Yaskawa INFORM job: X2_50&56B(90_180).JBI

/JOB
//NAME X2_50&56B(90_180)
//POS
///NPOS 380,380,380,17,0,0
///TOOL 0
///POSTYPE PULSE
///PULSE
C00000=45487,-81749,-76140,5313,88955,-2714
C00001=100725,-66680,-65098,5325,101088,31571
C00002=134065,-13803,-33339,15050,117611,54074
C00003=178572,20950,5765,5105,121785,76071
C00004=178477,15787,3727,4983,120398,75966
C00005=178438,13766,2992,4934,119816,75923
C00006=178435,14063,4928,4877,118781,75875
C00007=178438,13766,2992,4934,119816,75923
C00008=180168,17754,7052,5608,119256,76587
C00009=180168,18141,9405,5533,118013,76523
C00010=179359,16071,7488,5217,118182,76212
C00011=180168,18141,9405,5533,118013,76523
C00012=172189,10953,2801,14884,115134,86218
C00013=173139,8005,189,15209,115045,86581
C00014=172189,10953,2801,14884,115134,86218
C00015=169290,3234,-9196,14399,118965,85580
C00016=130973,-13523,-33423,14333,118859,53260
C00017=110700,-69385,-63067,6190,97747,34870
C00018=68653,-71679,-73408,24733,95794,85842
C00019=66615,-75998,-75470,24709,95531,75346
C00020=80537,-29900,-12555,12207,96591,80441
C00021=81172,-32243,-10721,12278,94215,80425
C00022=81559,-32147,-8308,12330,92754,80411
C00023=81559,-31652,-7175,12323,92320,80369
C00024=79890,-31226,-7999,11978,93276,79895
C00025=78854,-29246,-5136,11740,92696,79487
C00026=78019,-31526,-6644,11553,92575,79192
C00027=78854,-29246,-5136,11740,92696,79487
C00028=78535,-28461,-4244,11667,92599,79369
C00029=79905,-29828,-5160,11964,92267,79802
C00030=78535,-28461,-4244,11667,92599,79369
C00031=80655,-29539,-12313,12233,96610,80484
C00032=172905,9069,10368,17661,103953,63205
C00033=172925,6453,11622,17490,101927,62911
C00034=172953,5852,13232,17402,100678,62738
C00035=172980,6410,14735,17366,100062,62659
C00036=172934,5478,12205,17429,101103,62793
C00037=174868,12262,20269,17776,99277,63224
C00038=175653,10008,18253,17959,99184,63493
C00039=174868,12262,20269,17776,99277,63224
C00040=175466,10534,19114,17901,98978,63395
C00041=174549,8650,17530,17692,99183,63095
C00042=175466,10534,19114,17901,98978,63395
C00043=175364,13912,17144,18083,101810,63784
C00044=143557,-6058,-8183,20909,99706,63742
C00045=116076,-21395,-35361,8294,99864,-41660
C00046=116170,-16904,-19810,8141,92666,-42104
C00047=120850,-15711,-13213,8164,88779,-40753
C00048=120850,-15320,-11697,8164,88052,-40800
C00049=120850,-15603,-12792,8164,88575,-40767
C00050=118682,-15547,-12749,8147,88797,-41494
C00051=118682,-15195,-11396,8147,88151,-41535
C00052=119909,-15242,-11433,8154,88024,-41123
C00053=118283,-15171,-11379,8139,88193,-41669
C00054=118283,-17130,-20118,8163,92522,-41388
C00055=123081,10517,-9626,8350,99710,-39267
C00056=125078,45057,28923,8216,93591,-38991
C00057=129546,52045,50715,11678,83315,-38263
C00058=130769,54168,55563,11090,81346,-37992
C00059=131361,55704,59445,11868,79480,-38000
C00060=131361,56824,62095,11904,78446,-38101
C00061=127122,55959,62427,19640,78177,-40212
C00062=127429,56070,62553,19642,78085,-40116
C00063=127122,55959,62427,19640,78177,-40212
C00064=129532,54159,56872,13383,80275,-38621
C00065=128124,50047,46438,13290,84703,-38634
C00066=127892,65351,66100,15155,93024,-73666
C00067=127759,64877,68102,15105,91623,-73885
C00068=127759,66176,71014,15089,90535,-74019
C00069=127759,65952,70519,15092,90719,-73996
C00070=127818,62899,66930,15111,91326,-73901
C00071=127761,65124,68737,15102,91367,-73918
C00072=129268,64619,66746,9110,92510,-72857
C00073=129453,59738,62113,10172,92738,-72844
C00074=128543,59689,62492,12247,92447,-73324
C00075=129453,59738,62113,10172,92738,-72844
C00076=127856,24038,11624,3768,91984,-73094
C00077=122306,-16388,-19846,12665,86048,-29933
C00078=132420,-34549,-26934,9469,66215,-6029
C00079=130208,-34570,-23440,17968,63087,-6635
C00080=130112,-33170,-22523,17973,63257,-6644
C00081=130128,-33400,-22674,17972,63230,-6643
C00082=130128,-32836,-20938,18092,62486,-6765
C00083=130258,-35461,-24440,17930,63226,-6591
C00084=124734,-36329,-24999,19557,64397,-8564
C00085=124929,-32941,-19340,19786,62706,-8791
C00086=125915,-32833,-19269,19505,62482,-8438
C00087=124929,-32941,-19340,19786,62706,-8791
C00088=126330,-55457,-44088,9994,61079,1914
C00089=100312,-41100,-48322,7887,99302,-47123
C00090=117190,-44298,-39598,8136,90680,-41883
C00091=119238,-43364,-35384,8150,88380,-41331
C00092=120058,-42901,-33636,8158,87468,-41110
C00093=120057,-42457,-32093,8159,86753,-41157
C00094=120058,-42901,-33636,8158,87468,-41110
C00095=114736,-42040,-31696,13195,87643,-42975
C00096=115963,-42182,-31783,13219,87424,-42572
C00097=114736,-42040,-31696,13195,87643,-42975
C00098=113802,-42392,-33303,13175,88582,-43200
C00099=111477,-43037,-37156,13132,90949,-43758
C00100=102346,-51424,-37016,7803,86952,-47198
C00101=99301,-49115,-33281,12338,87461,-48360
C00102=100828,-48093,-29089,11211,84887,-48016
C00103=100828,-47667,-27999,11214,84443,-48056
C00104=100828,-48093,-29089,11211,84887,-48016
C00105=94654,-43932,-24417,16982,87204,-50251
C00106=95410,-44352,-24668,17050,86989,-50017
C00107=94654,-43932,-24417,16982,87204,-50251
C00108=98985,-47843,-30066,12603,86269,-48577
C00109=96616,-48227,-33817,12459,88698,-49151
C00110=47420,-68852,-70475,7734,99047,-48455
C00111=58856,-91847,-113443,3781,117020,-74641
C00112=60236,-59653,-81414,8514,109210,-81552
C00113=65712,-50088,-67931,3279,110982,-81026
C00114=65935,-54727,-66929,3231,107978,-81030
C00115=66231,-56054,-65409,3227,106352,-80970
C00116=66421,-55660,-64438,3238,105949,-80915
C00117=66309,-56041,-64890,3229,106036,-80952
C00118=66048,-59202,-66118,3188,105179,-81066
C00119=66309,-56041,-64890,3229,106036,-80952
C00120=65984,-49861,-66477,3286,110194,-80952
C00121=118683,-89548,-94864,-6316,107762,-74317
C00122=118830,-94736,-93309,-6169,104171,-74077
C00123=118897,-96147,-91968,-6116,102635,-73976
C00124=118911,-94939,-90367,-6104,102273,-73953
C00125=118926,-95247,-90740,-6105,102345,-73951
C00126=120069,-98591,-91538,-5957,101210,-73497
C00127=118926,-95247,-90740,-6105,102345,-73951
C00128=124253,-93200,-90530,-5582,103647,-72150
C00129=124297,-94887,-90828,-5558,102970,-72104
C00130=122332,-96938,-91342,-5745,102098,-72750
C00131=124297,-94887,-90828,-5558,102970,-72104
C00132=123836,-88068,-93172,-5765,107861,-72497
C00133=103947,-87224,-93768,11726,103256,-73456
C00134=105491,-91629,-91965,11598,99731,-73257
C00135=106242,-92046,-89539,11549,97951,-73163
C00136=106280,-91630,-88956,11545,97803,-73164
C00137=106194,-91849,-89665,11554,98133,-73164
C00138=106981,-95473,-90615,11530,96768,-73018
C00139=106194,-91849,-89665,11554,98133,-73164
C00140=107390,-94613,-90436,11549,97035,-72851
C00141=105229,-95826,-90624,11481,96844,-73620
C00142=107390,-94613,-90436,11549,97035,-72851
C00143=105129,-89034,-93253,11689,101866,-73178
C00144=117235,-90812,-97794,11932,101979,-68958
C00145=119184,-94938,-95823,11777,98434,-68628
C00146=119997,-95229,-93380,11717,96698,-68512
C00147=120000,-94762,-92745,11713,96550,-68526
C00148=120085,-95315,-93448,11717,96683,-68484
C00149=121254,-98780,-94295,11676,95281,-68213
C00150=120085,-95315,-93448,11717,96683,-68484
C00151=120732,-97303,-93959,11694,95897,-68335
C00152=122720,-95241,-93443,11703,96339,-67606
C00153=120732,-97303,-93959,11694,95897,-68335
C00154=117928,-92127,-96991,11873,100734,-68840
C00155=83815,-72409,-71600,49856,101385,-80874
C00156=86977,-76307,-70966,49554,98078,-81004
C00157=85918,-79626,-70912,49280,97499,-81857
C00158=85722,-81512,-70616,49126,96837,-82303
C00159=87678,-80975,-72090,49364,96559,-81447
C00160=88529,-80279,-70734,49348,95782,-81419
C00161=87018,-80378,-72384,49396,97246,-81423
C00162=92255,-82689,-76075,49623,95110,-79856
C00163=92255,-82357,-74554,49552,94603,-80124
C00164=91886,-84274,-76762,49584,95051,-80076
C00165=87038,-78982,-77882,49995,99948,-79968
C00166=111885,-94745,-96836,21175,93099,-57761
C00167=115356,-96241,-94167,20812,89966,-57066
C00168=116782,-95898,-92034,20669,88542,-56800
C00169=116805,-94979,-90810,20667,88272,-56838
C00170=117687,-92490,-90484,20584,89063,-56388
C00171=119638,-92586,-90524,20383,88555,-55777
C00172=116782,-95072,-90979,20669,88331,-56836
C00173=116675,-98914,-91892,20684,87033,-57096
C00174=116782,-95072,-90979,20669,88331,-56836
C00175=111949,-93327,-94846,21154,92619,-57823
C00176=55380,-134082,-104834,55812,75253,-81172
C00177=61753,-134169,-102482,55825,70609,-80463
C00178=64815,-132350,-99998,55791,68452,-80067
C00179=65073,-131468,-99170,55790,68267,-80036
C00180=65012,-131683,-99347,55795,68302,-80050
C00181=67421,-134585,-100123,55949,66292,-79958
C00182=65012,-131683,-99347,55795,68302,-80050
C00183=66833,-133758,-99865,55902,66793,-79972
C00184=68699,-130981,-99713,55278,66469,-79035
C00185=66833,-133758,-99865,55902,66793,-79972
C00186=57706,-134492,-103408,55942,73242,-81128
C00187=64785,-112873,-118243,24954,102118,-81978
C00188=94326,-86621,-83484,-35338,109503,-87169
C00189=91634,-91881,-83017,-35113,105930,-87131
C00190=90294,-93871,-83332,-35163,104694,-87298
C00191=90673,-91662,-79967,-34941,104076,-86932
C00192=96279,-95614,-77654,-39133,100534,-74699
C00193=97530,-94207,-78400,-39125,102027,-74707
C00194=99906,-89889,-79610,-39309,105429,-74936
C00195=93707,-90060,-101982,-2678,109676,-68403
C00196=85859,-88563,-85007,37375,108858,-60120
C00197=89767,-92929,-84612,37372,105169,-59726
C00198=92261,-92553,-83552,37602,103718,-59151
C00199=87809,-89294,-77804,36664,104133,-60948
C00200=97825,-97090,-85633,28728,98264,-58810
C00201=105101,-94972,-90460,21721,102166,-53461
C00202=101619,-91841,-92201,21697,105576,-54126
C00203=110011,-90138,-98551,28023,73725,-47627
C00204=114073,-86949,-94757,26595,71811,-46539
C00205=115509,-85532,-93350,26060,71244,-46123
C00206=116669,-38852,-76477,24599,105061,-42370
C00207=113194,-138803,-104651,24561,74823,-49786
C00208=115868,-123842,-100277,21543,88201,-42617
C00209=113813,-124047,-101616,21486,89414,-43150
C00210=108993,-124666,-104884,21332,92253,-44397
C00211=109211,-98340,-98499,17204,97884,-65653
C00212=111963,-101539,-96259,17038,94417,-65168
C00213=114319,-101452,-95162,16976,93323,-64488
C00214=121130,-95827,-93982,7505,98794,-69297
C00215=120137,-94785,-95042,7509,100063,-69562
C00216=118600,-90390,-96949,7580,103607,-69872
C00217=87744,-101201,-89183,32285,100120,-63549
C00218=91822,-104522,-87796,32421,96378,-62986
C00219=93007,-105888,-87219,32449,95024,-62902
C00220=125171,-100001,-94421,10746,96250,-68519
C00221=112189,-112791,-97117,10082,92847,-73286
C00222=125737,-104595,-94231,123,98676,-80328
C00223=125012,-83838,-85262,564,111182,-80520
C00224=124880,-77934,-85992,554,114665,-80551
C00225=118378,-61430,-80227,-500,113656,-60542
C00226=119635,-65792,-78782,-346,110532,-60082
C00227=120344,-67374,-78220,-265,109375,-59827
C00228=117636,-69991,-79065,-562,108539,-60782
C00229=61499,-79673,-75485,-5801,99043,-80116
C00230=59682,-78713,-74784,-5933,98973,-80740
C00231=58729,-76685,-75165,-6027,100171,-81128
C00232=59096,-71470,-86943,-6341,110071,-81508
C00233=60236,-59653,-81414,8514,109210,-81552
C00234=58856,-91847,-113443,3781,117020,-74641
C00235=47420,-68852,-70475,7734,99047,-48455
C00236=126000,-95797,-97639,-7032,71909,3420
C00237=125334,-73481,-62420,-7403,61720,3825
C00238=136814,-5072,7481,118,87452,82611
C00239=137691,-48649,-34753,2434,90887,80546
C00240=137775,-50281,-31902,2439,88294,80524
C00241=138073,-51533,-31005,2464,87091,80603
C00242=135282,-52527,-31425,2223,86909,79659
C00243=133173,-53016,-31621,2042,86835,78950
C00244=130291,-53529,-31930,1793,86840,77980
C00245=130424,-52342,-33062,1804,88142,78044
C00246=109921,-30503,-12357,16555,100596,88828
C00247=106221,-34483,-13308,18126,97869,90694
C00248=105952,-33586,-11090,18011,97063,90477
C00249=105952,-33586,-11090,18011,97063,90477
C00250=108084,-28000,-11018,16080,101404,88284
C00251=146524,-12798,-32,-1632,107432,69723
C00252=150731,-18568,-2319,-5233,105441,66132
C00253=150931,-18182,-1503,-5155,105151,66214
C00254=151130,-17517,-94,-5073,104642,66304
C00255=149548,-12799,1040,-3936,106552,67422
C00256=137932,-46455,-34045,2456,91570,80642
C00257=130584,-47998,-33152,21701,103265,82699
C00258=131924,-51228,-32028,21814,100720,82725
C00259=132596,-53048,-31639,21886,99448,82739
C00260=136106,-52307,-31332,22746,98680,83888
C00261=136106,-52307,-31332,22746,98680,83888
C00262=136106,-52307,-31332,22746,98680,83888
C00263=135156,-50442,-31749,22619,100068,83801
C00264=145953,-54402,-37679,17502,96627,81619
C00265=151175,-48657,-29446,15262,96856,77657
C00266=143727,-65526,-38899,20404,85578,88618
C00267=138380,-68197,-47605,21119,89179,90269
C00268=135468,-61779,-51499,19715,96090,83313
C00269=146504,11659,2252,17659,107540,74925
C00270=144153,-20650,-13732,15502,93070,-1402
C00271=144800,-23297,881,19511,75808,-35743
C00272=150747,-18290,7168,14784,74611,-33299
C00273=151238,-17498,8369,14810,74204,-33179
C00274=149375,-28253,2716,19877,71272,-34860
C00275=147327,-9055,19175,22000,84077,-38130
C00276=145889,24730,54854,22060,94685,-42086
C00277=143819,24834,51946,21414,96917,-42392
C00278=152079,-13657,11289,11329,66320,-30599
C00279=154406,-11055,15215,8681,65213,-29600
C00280=152146,-117,24134,8927,65583,-30385
C00281=151595,-2013,20658,8910,66792,-30489
C00282=149654,-12806,15500,15951,62742,-32403
C00283=154253,-10520,16648,9945,64198,-29883
C00284=152115,-1183,24071,10179,64683,-30617
C00285=151630,-3056,20389,10130,66025,-30671
C00286=149245,-3141,19709,11821,66260,-31671
C00287=148434,-2355,21995,13515,64976,-32267
C00288=147463,3367,26836,13655,65100,-32622
C00289=153331,-4155,20539,5600,59410,-15455
C00290=155287,-19713,9431,3047,50741,-18387
C00291=157786,-39099,-6604,-901,42168,-20790
C00292=135242,-54877,-19518,11584,43472,-31405
C00293=131236,-19596,-17600,13529,71052,-30429
C00294=140706,-23702,-4175,12836,48543,-13474
C00295=140673,-21200,-1486,12925,48190,-13534
C00296=141284,-13369,5846,23551,49891,-17686
C00297=139681,-13144,7389,23829,50519,-19910
C00298=143196,-11606,9882,18412,48184,-18316
C00299=142607,-11156,11441,21979,47155,-19159
C00300=141350,-14076,4076,20421,51470,-19989
C00301=145280,-15693,1343,3360,54502,-7889
C00302=146672,-15493,4014,938,50764,-7216
C00303=145826,-15296,5401,6578,48621,-8155
C00304=140850,-20387,-3678,6927,53662,-12969
C00305=114161,26367,33601,23969,88215,-55914
C00306=115200,37711,50954,30924,91004,-62691
C00307=115095,42493,60117,30863,88292,-63457
C00308=111984,51906,52240,30690,97793,-62104
C00309=127032,55270,53918,12904,96771,-63979
C00310=128416,55540,54262,13146,96476,-63525
C00311=127174,62998,65861,21032,96181,-64334
C00312=128287,63468,66410,21260,95807,-63997
C00313=128287,63468,66410,21260,95807,-63997
C00314=127978,65974,69378,21169,95383,-64184
C00315=127955,65548,69421,21154,95160,-64232
C00316=128682,65721,69556,21305,94980,-64002
C00317=120314,64980,62876,19697,100558,-66081
C00318=132001,51753,30880,19285,94077,-28834
C00319=133943,71841,58405,19142,87355,-29202
C00320=134114,75534,69283,19228,82775,-29864
C00321=134337,77934,74847,17635,80860,-30005
C00322=135526,64406,59304,14794,72965,-27180
C00323=135838,44640,35862,12862,72937,-25659
C00324=131873,33832,21789,16508,74721,-32134
C00325=132107,40218,30480,18908,92419,-37660
C00326=132579,41227,34664,18882,90360,-37810
C00327=134167,43289,37766,16302,89928,-37295
C00328=135380,31026,24943,15599,91467,-36659
C00329=134217,44561,36967,16470,93837,-37645
C00330=131769,55424,45596,17778,98765,-39318
C00331=127656,48680,32292,16283,104912,-42086
C00332=116663,7338,4481,17873,88938,-41861
C00333=82713,25471,38030,41323,96034,-53690
C00334=86390,18515,43854,41800,88900,-54935
C00335=84848,25261,59330,49223,87350,-55843
C00336=88606,53039,89487,50588,82672,-56584
C00337=87361,53333,88208,50128,83897,-56499
C00338=87606,32039,49279,49923,92343,-51642
C00339=120401,-109118,-96895,24846,84275,-3219
C00340=171543,-75667,-77525,-32488,107850,47798
C00341=131110,-7914,-12100,-23259,79386,39340
C00342=129844,-3252,1633,-26699,74465,49623
C00343=129212,9628,12610,-26630,74140,49455
C00344=129658,-2563,931,-26586,75112,49402
C00345=129658,-2563,931,-26586,75112,49402
C00346=129347,-1591,2560,-26600,74559,49410
C00347=128897,8094,10886,-26554,74283,49298
C00348=136882,-16782,-14142,-32633,69855,42519
C00349=146203,-27363,-23504,-26744,90214,39705
C00350=126939,-13199,-3011,-17863,102554,59788
C00351=123418,-15871,2353,-18433,97326,59310
C00352=121177,-12096,8576,-18692,97429,62482
C00353=122121,-11145,10388,-18399,97041,62873
C00354=122578,-10954,11934,-18230,96330,63143
C00355=117631,-18242,3340,-13059,93114,62902
C00356=122301,-18046,-869,-17501,95215,65467
C00357=137808,-17234,-5965,-14129,101643,70132
C00358=160865,-72571,-62696,-26432,95765,43985
C00359=33343,-40499,-55087,21473,103101,25780
C00360=36142,-38032,-53479,26160,91217,55204
C00361=34841,-42177,-53650,26305,89793,54410
C00362=37290,-39771,-48911,25965,87520,54810
C00363=53650,-84621,-72547,23787,74875,58246
C00364=53650,-84621,-72547,23787,74875,58246
C00365=51472,-81480,-75734,23883,78787,58225
C00366=145140,-22572,-14465,18960,94137,68113
C00367=156171,-3243,9823,12083,101691,63095
C00368=154843,-3158,11434,13995,99637,65375
C00369=156075,-1201,14334,13752,98988,65034
C00370=157211,1579,14506,12356,101141,63409
C00371=145375,-16597,89,21780,91791,76946
C00372=153486,-12500,3434,13683,93075,81038
C00373=153486,-12500,3434,13683,93075,81038
C00374=145663,-7270,12633,24862,92938,88979
C00375=142776,-6009,11285,24301,95132,88379
C00376=125886,-7477,896,20570,104940,83992
C00377=123761,-17662,-8863,23291,102823,83503
C00378=103503,-37411,-26995,22689,104461,77175
C00379=-2000,-113393,-91320,0,88983,0
BC00000=213476,520800,586713
BC00001=246976,521618,248910
BC00002=313048,446954,225880
BC00003=365345,432483,248910
BC00004=365345,432483,248910
BC00005=365345,432483,248910
BC00006=365345,432483,248910
BC00007=365345,432483,248910
BC00008=365345,432483,248910
BC00009=365345,432483,248910
BC00010=365345,432483,248910
BC00011=365345,432483,248910
BC00012=365345,432483,248910
BC00013=365345,432483,248910
BC00014=365345,432483,248910
BC00015=365345,432483,248910
BC00016=315213,470551,248910
BC00017=253462,521618,248910
BC00018=74243,523374,420920
BC00019=74243,435039,420920
BC00020=74243,435039,420920
BC00021=74243,435039,420920
BC00022=74243,435039,420920
BC00023=74243,435039,420920
BC00024=74243,435039,420920
BC00025=74243,435039,420920
BC00026=74243,435039,420920
BC00027=74243,435039,420920
BC00028=74243,435039,420920
BC00029=74243,435039,420920
BC00030=74243,435039,420920
BC00031=74243,435039,420920
BC00032=168837,433490,369354
BC00033=168837,433490,369354
BC00034=168837,435026,369354
BC00035=168837,435026,369354
BC00036=168837,435026,369354
BC00037=168837,435026,369354
BC00038=168837,435026,369354
BC00039=168837,435026,369354
BC00040=168837,435026,369354
BC00041=168837,435026,369354
BC00042=168837,435026,369354
BC00043=168837,435026,369354
BC00044=153053,422718,383276
BC00045=133884,399020,347416
BC00046=133886,399021,347410
BC00047=133886,399021,347410
BC00048=133886,399021,347410
BC00049=133886,399021,347410
BC00050=133886,399021,347410
BC00051=133886,399021,347410
BC00052=133886,399021,347410
BC00053=133886,399021,347410
BC00054=133886,399021,347410
BC00055=133884,399020,347416
BC00056=102028,399020,347416
BC00057=99639,399020,347416
BC00058=99639,399020,347416
BC00059=99639,399020,347416
BC00060=99639,399020,347416
BC00061=99639,399020,347416
BC00062=99639,399020,347416
BC00063=99639,399020,347416
BC00064=99639,399020,347416
BC00065=99639,399020,347416
BC00066=99639,399020,347415
BC00067=99639,399020,347415
BC00068=99639,399020,347415
BC00069=99639,399020,347415
BC00070=99639,399020,347415
BC00071=99639,399020,347415
BC00072=99639,399020,347415
BC00073=99639,399020,347415
BC00074=99639,399020,347415
BC00075=99639,399020,347415
BC00076=99639,399020,347415
BC00077=99639,399020,347415
BC00078=99638,399020,347413
BC00079=99638,399020,347413
BC00080=99638,399020,347413
BC00081=99638,399020,347413
BC00082=99638,399020,347413
BC00083=99638,399020,347413
BC00084=99638,399020,347413
BC00085=99638,399020,347413
BC00086=99638,399020,347413
BC00087=99638,399020,347413
BC00088=99638,399020,347413
BC00089=57428,399020,305871
BC00090=57428,399020,305871
BC00091=57428,399020,305871
BC00092=57428,399020,305871
BC00093=57428,399020,305871
BC00094=57428,399020,305871
BC00095=57428,399020,305871
BC00096=57428,399020,305871
BC00097=57428,399020,305871
BC00098=57428,399020,305871
BC00099=57428,399020,305871
BC00100=31464,452158,350496
BC00101=31464,452158,350496
BC00102=31464,452158,350496
BC00103=31464,452158,350496
BC00104=31464,452158,350496
BC00105=31464,452158,350496
BC00106=31464,452158,350496
BC00107=31464,452158,350496
BC00108=31464,452158,350496
BC00109=31464,452158,350496
BC00110=45599,519934,524307
BC00111=269547,451113,1075193
BC00112=398158,407689,1075139
BC00113=398158,407689,1075139
BC00114=398158,407689,1075139
BC00115=398158,406460,1075139
BC00116=398158,406460,1075139
BC00117=398158,406460,1075139
BC00118=398158,406460,1075139
BC00119=398158,406460,1075139
BC00120=398158,406460,1075139
BC00121=387339,358578,1075139
BC00122=387339,358578,1075139
BC00123=387339,358578,1075139
BC00124=387339,358578,1075139
BC00125=387339,358578,1075139
BC00126=387339,358578,1075139
BC00127=387339,358578,1075139
BC00128=387339,358578,1075139
BC00129=387339,358578,1075139
BC00130=387339,358578,1075139
BC00131=387339,358578,1075139
BC00132=387339,358578,1075139
BC00133=398158,372129,1075139
BC00134=398158,372129,1075139
BC00135=398158,372129,1075139
BC00136=398158,372129,1075139
BC00137=398158,372129,1075139
BC00138=398158,372129,1075139
BC00139=398158,372129,1075139
BC00140=398158,372129,1075139
BC00141=398158,372129,1075139
BC00142=398158,372129,1075139
BC00143=398158,372129,1075139
BC00144=394158,359189,1075139
BC00145=394158,359189,1075139
BC00146=394158,359189,1075139
BC00147=394158,359189,1075139
BC00148=394158,359189,1075139
BC00149=394158,359189,1075139
BC00150=394158,359189,1075139
BC00151=394158,359189,1075139
BC00152=394158,359189,1075139
BC00153=394158,359189,1075139
BC00154=394158,359189,1075139
BC00155=398158,378660,1075139
BC00156=398158,378660,1075139
BC00157=398158,378660,1075139
BC00158=398158,378660,1075139
BC00159=398158,378660,1075139
BC00160=398158,378660,1075139
BC00161=398158,378660,1075139
BC00162=398158,378660,1075139
BC00163=398158,378660,1075139
BC00164=398158,378660,1075139
BC00165=398158,378660,1075139
BC00166=398158,368832,1075139
BC00167=398158,368832,1075139
BC00168=398158,368832,1075139
BC00169=398158,368832,1075139
BC00170=398158,368832,1075139
BC00171=398158,368832,1075139
BC00172=398158,368832,1075139
BC00173=398158,368832,1075139
BC00174=398158,368832,1075139
BC00175=398158,368832,1075139
BC00176=357517,306686,1075139
BC00177=357517,306686,1075139
BC00178=357517,306686,1075139
BC00179=357517,306686,1075139
BC00180=357517,306686,1075139
BC00181=357517,306686,1075139
BC00182=357517,306686,1075139
BC00183=357517,306686,1075139
BC00184=357517,306686,1075139
BC00185=357517,306686,1075139
BC00186=357517,306686,1075139
BC00187=340869,312184,1075139
BC00188=309744,322463,1075139
BC00189=309744,322463,1075139
BC00190=309744,322463,1075139
BC00191=309744,322463,1075139
BC00192=309744,322463,1075139
BC00193=309744,322463,1075139
BC00194=309744,322463,1075139
BC00195=346127,336854,1075139
BC00196=394153,355850,1075139
BC00197=394153,355850,1075139
BC00198=394153,355850,1075139
BC00199=394153,355850,1075139
BC00200=394153,355850,1075139
BC00201=394153,355850,1075139
BC00202=394153,355850,1075139
BC00203=398158,337719,1075139
BC00204=398158,337719,1075139
BC00205=398158,337719,1075139
BC00206=398158,337719,1075139
BC00207=398158,337719,1075139
BC00208=398158,337719,1075139
BC00209=398158,337719,1075139
BC00210=398158,337719,1075139
BC00211=383630,353340,1075139
BC00212=383630,353340,1075139
BC00213=383631,353339,1075138
BC00214=383630,353340,1075139
BC00215=383630,353340,1075139
BC00216=383630,353340,1075139
BC00217=398158,354245,1075139
BC00218=398158,354245,1075139
BC00219=398158,354245,1075139
BC00220=398158,354245,1075139
BC00221=398158,354245,1075139
BC00222=398158,354245,1075139
BC00223=398158,354245,1075139
BC00224=398158,354245,1075139
BC00225=398158,383071,1075139
BC00226=398158,383071,1075139
BC00227=398158,383071,1075139
BC00228=398158,383071,1075139
BC00229=398158,383071,1075139
BC00230=398158,383071,1075139
BC00231=398158,383071,1075139
BC00232=398158,383071,1075139
BC00233=398158,407689,1075139
BC00234=269547,451113,1075193
BC00235=45599,519934,524307
BC00236=94263,511214,315317
BC00237=94263,460396,315317
BC00238=135587,422824,502968
BC00239=127942,440744,374117
BC00240=127942,440744,374117
BC00241=127942,440744,374117
BC00242=127942,440744,374117
BC00243=127942,440744,374117
BC00244=127942,440744,374117
BC00245=127942,440744,374117
BC00246=127942,440744,374117
BC00247=127942,440744,374117
BC00248=127942,440744,374117
BC00249=127942,440744,374117
BC00250=127942,440744,374117
BC00251=127942,440744,374117
BC00252=127942,440744,374117
BC00253=127942,440744,374117
BC00254=127942,440744,374117
BC00255=127942,440744,374117
BC00256=127942,440744,374117
BC00257=104807,412877,320931
BC00258=104807,412877,320931
BC00259=104807,412877,320931
BC00260=104807,412877,320931
BC00261=104807,412877,320931
BC00262=104807,412877,320931
BC00263=104807,412877,320931
BC00264=104807,412877,320931
BC00265=104807,412877,320931
BC00266=104807,412877,320931
BC00267=104807,412877,320931
BC00268=104807,412877,320931
BC00269=148089,457110,367423
BC00270=136783,454432,423186
BC00271=131867,453267,447430
BC00272=131867,453267,447430
BC00273=131867,453267,447430
BC00274=131867,453267,447430
BC00275=131867,453267,447430
BC00276=131867,453267,447430
BC00277=131867,453267,447430
BC00278=135848,460777,463714
BC00279=135848,460777,463714
BC00280=135848,460777,463714
BC00281=135848,460777,463714
BC00282=135930,434945,463100
BC00283=135941,432529,463037
BC00284=135941,432529,463037
BC00285=135941,432529,463037
BC00286=132949,418332,450445
BC00287=132950,418333,450445
BC00288=132950,418333,450445
BC00289=132950,418333,450445
BC00290=132950,418333,450445
BC00291=132949,418332,450445
BC00292=132949,418332,450445
BC00293=129700,411017,399742
BC00294=129700,411017,399742
BC00295=129700,411017,399742
BC00296=129700,411017,399742
BC00297=129700,411017,399742
BC00298=129700,411017,399742
BC00299=129700,411017,399742
BC00300=129700,411017,399742
BC00301=129700,411017,399742
BC00302=129700,411017,399742
BC00303=129700,411017,399742
BC00304=129700,411017,399742
BC00305=93339,398780,399742
BC00306=97844,394978,399742
BC00307=97844,394978,399742
BC00308=97844,394978,319091
BC00309=97844,394978,319091
BC00310=97844,394978,319091
BC00311=97844,394978,319091
BC00312=97844,394978,319091
BC00313=97844,394978,319091
BC00314=97844,394978,319091
BC00315=97844,394978,319091
BC00316=97844,394978,319091
BC00317=97844,394978,319091
BC00318=124371,399020,235938
BC00319=124371,400539,247766
BC00320=124371,400539,247766
BC00321=122136,400544,260322
BC00322=122136,400544,260322
BC00323=118659,400548,263238
BC00324=114198,400554,266980
BC00325=113920,399020,281296
BC00326=113920,399020,281296
BC00327=113920,399020,281296
BC00328=113921,399022,281295
BC00329=113921,399021,281295
BC00330=113920,399020,281296
BC00331=113920,399020,281296
BC00332=116853,417006,397633
BC00333=116853,417006,397633
BC00334=116853,417006,397633
BC00335=116853,417006,397633
BC00336=116853,417006,397633
BC00337=116853,417006,397633
BC00338=116980,417784,398351
BC00339=133964,521927,494526
BC00340=6376,521927,323535
BC00341=801,413740,323535
BC00342=801,409504,323535
BC00343=801,409504,323535
BC00344=801,409504,323535
BC00345=801,409504,323535
BC00346=801,409504,323535
BC00347=801,409504,323535
BC00348=801,404489,323535
BC00349=6376,456068,397764
BC00350=6376,456068,397764
BC00351=6376,456068,397764
BC00352=5796,456884,400752
BC00353=6376,457056,399834
BC00354=6376,456068,402258
BC00355=6376,456068,399147
BC00356=6376,456068,397764
BC00357=6376,456068,397764
BC00358=6376,515380,482255
BC00359=159570,501423,294766
BC00360=173097,444830,189232
BC00361=173097,444830,189232
BC00362=173097,444830,189232
BC00363=173097,444830,189232
BC00364=173097,444830,189232
BC00365=173097,444830,189232
BC00366=325503,445921,382394
BC00367=329528,445950,387496
BC00368=329528,445950,387496
BC00369=329528,445950,387496
BC00370=329528,445950,387496
BC00371=329528,445950,387496
BC00372=329528,445950,387496
BC00373=329528,445950,387496
BC00374=329528,445950,387496
BC00375=329528,445950,387496
BC00376=299842,445950,387496
BC00377=298777,512077,364490
BC00378=247805,558426,416413
BC00379=87173,523905,1075193
EC00000=-798156,-1296783
EC00001=-798156,-1296783
EC00002=-798156,-1296783
EC00003=-798156,-1296783
EC00004=-798156,-1296783
EC00005=-798156,-1296783
EC00006=-798156,-1296783
EC00007=-798156,-1296783
EC00008=-798156,-1296783
EC00009=-798156,-1296783
EC00010=-798156,-1296783
EC00011=-798156,-1296783
EC00012=-798156,-1296783
EC00013=-798156,-1296783
EC00014=-798156,-1296783
EC00015=-798156,-1296783
EC00016=-798156,-1296783
EC00017=-798156,-1296783
EC00018=-798156,-1296783
EC00019=-798156,-1296783
EC00020=-798156,-1296783
EC00021=-798156,-1296783
EC00022=-798156,-1296783
EC00023=-798156,-1296783
EC00024=-798156,-1296783
EC00025=-798156,-1296783
EC00026=-798156,-1296783
EC00027=-798156,-1296783
EC00028=-798156,-1296783
EC00029=-798156,-1296783
EC00030=-798156,-1296783
EC00031=-798156,-1296783
EC00032=-798156,-1296783
EC00033=-798156,-1296783
EC00034=-798156,-1296783
EC00035=-798156,-1296783
EC00036=-798156,-1296783
EC00037=-798156,-1296783
EC00038=-798156,-1296783
EC00039=-798156,-1296783
EC00040=-798156,-1296783
EC00041=-798156,-1296783
EC00042=-798156,-1296783
EC00043=-798156,-1296783
EC00044=-798156,-1296783
EC00045=-798156,-1296783
EC00046=-798154,-1296781
EC00047=-798154,-1296781
EC00048=-798154,-1296781
EC00049=-798154,-1296781
EC00050=-798154,-1296781
EC00051=-798154,-1296781
EC00052=-798154,-1296781
EC00053=-798154,-1296781
EC00054=-798154,-1296781
EC00055=-798156,-1296783
EC00056=-798156,-1296783
EC00057=-798156,-1296783
EC00058=-798156,-1296783
EC00059=-798156,-1296783
EC00060=-798156,-1296783
EC00061=-798156,-1296783
EC00062=-798156,-1296783
EC00063=-798156,-1296783
EC00064=-798156,-1296783
EC00065=-798156,-1296783
EC00066=-798155,-1296781
EC00067=-798155,-1296781
EC00068=-798155,-1296781
EC00069=-798155,-1296781
EC00070=-798155,-1296781
EC00071=-798155,-1296781
EC00072=-798155,-1296781
EC00073=-798155,-1296781
EC00074=-798155,-1296781
EC00075=-798155,-1296781
EC00076=-798155,-1296781
EC00077=-798155,-1296781
EC00078=-798154,-1296780
EC00079=-798154,-1296780
EC00080=-798154,-1296780
EC00081=-798154,-1296780
EC00082=-798154,-1296780
EC00083=-798154,-1296780
EC00084=-798154,-1296780
EC00085=-798154,-1296780
EC00086=-798154,-1296780
EC00087=-798154,-1296780
EC00088=-798154,-1296780
EC00089=-798156,-1296783
EC00090=-798156,-1296783
EC00091=-798156,-1296783
EC00092=-798156,-1296783
EC00093=-798156,-1296783
EC00094=-798156,-1296783
EC00095=-798156,-1296783
EC00096=-798156,-1296783
EC00097=-798156,-1296783
EC00098=-798156,-1296783
EC00099=-798156,-1296783
EC00100=-798156,-1296783
EC00101=-798156,-1296783
EC00102=-798156,-1296783
EC00103=-798156,-1296783
EC00104=-798156,-1296783
EC00105=-798156,-1296783
EC00106=-798156,-1296783
EC00107=-798156,-1296783
EC00108=-798156,-1296783
EC00109=-798156,-1296783
EC00110=-798156,-1296783
EC00111=-906908,-1296783
EC00112=-975524,-1296783
EC00113=-975524,-1296783
EC00114=-975524,-1296783
EC00115=-975524,-1296783
EC00116=-975524,-1296783
EC00117=-975524,-1296783
EC00118=-975524,-1296783
EC00119=-975524,-1296783
EC00120=-975524,-1296783
EC00121=-975524,-1296783
EC00122=-975524,-1296783
EC00123=-975524,-1296783
EC00124=-975524,-1296783
EC00125=-975524,-1296783
EC00126=-975524,-1296783
EC00127=-975524,-1296783
EC00128=-975524,-1296783
EC00129=-975524,-1296783
EC00130=-975524,-1296783
EC00131=-975524,-1296783
EC00132=-975524,-1296783
EC00133=-975524,-1296783
EC00134=-975524,-1296783
EC00135=-975524,-1296783
EC00136=-975524,-1296783
EC00137=-975524,-1296783
EC00138=-975524,-1296783
EC00139=-975524,-1296783
EC00140=-975524,-1296783
EC00141=-975524,-1296783
EC00142=-975524,-1296783
EC00143=-975524,-1296783
EC00144=-975524,-1296783
EC00145=-975524,-1296783
EC00146=-975524,-1296783
EC00147=-975524,-1296783
EC00148=-975524,-1296783
EC00149=-975524,-1296783
EC00150=-975524,-1296783
EC00151=-975524,-1296783
EC00152=-975524,-1296783
EC00153=-975524,-1296783
EC00154=-975524,-1296783
EC00155=-975524,-1296783
EC00156=-975524,-1296783
EC00157=-975524,-1296783
EC00158=-975524,-1296783
EC00159=-975524,-1296783
EC00160=-975524,-1296783
EC00161=-975524,-1296783
EC00162=-975524,-1296783
EC00163=-975524,-1296783
EC00164=-975524,-1296783
EC00165=-975524,-1296783
EC00166=-975524,-1296783
EC00167=-975524,-1296783
EC00168=-975524,-1296783
EC00169=-975524,-1296783
EC00170=-975524,-1296783
EC00171=-975524,-1296783
EC00172=-975524,-1296783
EC00173=-975524,-1296783
EC00174=-975524,-1296783
EC00175=-975524,-1296783
EC00176=-975524,-1296783
EC00177=-975524,-1296783
EC00178=-975524,-1296783
EC00179=-975524,-1296783
EC00180=-975524,-1296783
EC00181=-975524,-1296783
EC00182=-975524,-1296783
EC00183=-975524,-1296783
EC00184=-975524,-1296783
EC00185=-975524,-1296783
EC00186=-975524,-1296783
EC00187=-975524,-1296783
EC00188=-975524,-1296783
EC00189=-975524,-1296783
EC00190=-975524,-1296783
EC00191=-975524,-1296783
EC00192=-975524,-1296783
EC00193=-975524,-1296783
EC00194=-975524,-1296783
EC00195=-975524,-1296783
EC00196=-975524,-1296783
EC00197=-975524,-1296783
EC00198=-975524,-1296783
EC00199=-975524,-1296783
EC00200=-975524,-1296783
EC00201=-975524,-1296783
EC00202=-975524,-1296783
EC00203=-975524,-1296783
EC00204=-975524,-1296783
EC00205=-975524,-1296783
EC00206=-975524,-1296783
EC00207=-975524,-1296783
EC00208=-975524,-1296783
EC00209=-975524,-1296783
EC00210=-975524,-1296783
EC00211=-975524,-1296783
EC00212=-975524,-1296783
EC00213=-975522,-1296782
EC00214=-975524,-1296783
EC00215=-975524,-1296783
EC00216=-975524,-1296783
EC00217=-975524,-1296783
EC00218=-975524,-1296783
EC00219=-975524,-1296783
EC00220=-975524,-1296783
EC00221=-975524,-1296783
EC00222=-975524,-1296783
EC00223=-975524,-1296783
EC00224=-975524,-1296783
EC00225=-975524,-1296783
EC00226=-975524,-1296783
EC00227=-975524,-1296783
EC00228=-975524,-1296783
EC00229=-975524,-1296783
EC00230=-975524,-1296783
EC00231=-975524,-1296783
EC00232=-975524,-1296783
EC00233=-975524,-1296783
EC00234=-906908,-1296783
EC00235=-798156,-1296783
EC00236=-798156,-1296783
EC00237=-798156,-1296783
EC00238=-798156,-1296783
EC00239=-798156,-1296783
EC00240=-798156,-1296783
EC00241=-798156,-1296783
EC00242=-798156,-1296783
EC00243=-798156,-1296783
EC00244=-798156,-1296783
EC00245=-798156,-1296783
EC00246=-798156,-1296783
EC00247=-798156,-1296783
EC00248=-798156,-1296783
EC00249=-798156,-1296783
EC00250=-798156,-1296783
EC00251=-798156,-1296783
EC00252=-798156,-1296783
EC00253=-798156,-1296783
EC00254=-798156,-1296783
EC00255=-798156,-1296783
EC00256=-798156,-1296783
EC00257=-798156,-1296783
EC00258=-798156,-1296783
EC00259=-798156,-1296783
EC00260=-798156,-1296783
EC00261=-798156,-1296783
EC00262=-798156,-1296783
EC00263=-798156,-1296783
EC00264=-798156,-1296783
EC00265=-798156,-1296783
EC00266=-798156,-1296783
EC00267=-798156,-1296783
EC00268=-798156,-1296783
EC00269=-798156,-1296783
EC00270=-798156,-1296783
EC00271=-798156,-1296783
EC00272=-798156,-1296783
EC00273=-798156,-1296783
EC00274=-798156,-1296783
EC00275=-798156,-1296783
EC00276=-798156,-1296783
EC00277=-798156,-1296783
EC00278=-798156,-1296783
EC00279=-798156,-1296783
EC00280=-798156,-1296783
EC00281=-798156,-1296783
EC00282=-798153,-1296781
EC00283=-798156,-1296783
EC00284=-798156,-1296783
EC00285=-798156,-1296783
EC00286=-798156,-1296783
EC00287=-798155,-1296782
EC00288=-798155,-1296782
EC00289=-798155,-1296782
EC00290=-798155,-1296782
EC00291=-798156,-1296783
EC00292=-798156,-1296783
EC00293=-798156,-1296783
EC00294=-798156,-1296783
EC00295=-798156,-1296783
EC00296=-798156,-1296783
EC00297=-798156,-1296783
EC00298=-798156,-1296783
EC00299=-798156,-1296783
EC00300=-798156,-1296783
EC00301=-798156,-1296783
EC00302=-798156,-1296783
EC00303=-798156,-1296783
EC00304=-798156,-1296783
EC00305=-798156,-1296783
EC00306=-798156,-1296783
EC00307=-798156,-1296783
EC00308=-798156,-1296783
EC00309=-798156,-1296783
EC00310=-798156,-1296783
EC00311=-798156,-1296783
EC00312=-798156,-1296783
EC00313=-798156,-1296783
EC00314=-798156,-1296783
EC00315=-798156,-1296783
EC00316=-798156,-1296783
EC00317=-798156,-1296783
EC00318=-798156,-1296783
EC00319=-798156,-1296783
EC00320=-798156,-1296783
EC00321=-798156,-1296783
EC00322=-798156,-1296783
EC00323=-798156,-1296783
EC00324=-798156,-1296783
EC00325=-798156,-1296783
EC00326=-798156,-1296783
EC00327=-798156,-1296783
EC00328=-798154,-1296780
EC00329=-798154,-1296781
EC00330=-798156,-1296783
EC00331=-798156,-1296783
EC00332=-798156,-1296783
EC00333=-798156,-1296783
EC00334=-798156,-1296783
EC00335=-798156,-1296783
EC00336=-798156,-1296783
EC00337=-798156,-1296783
EC00338=-798156,-1296783
EC00339=-798156,-1296783
EC00340=-798156,-1296783
EC00341=-798156,-1296783
EC00342=-798156,-1296783
EC00343=-798156,-1296783
EC00344=-798156,-1296783
EC00345=-798156,-1296783
EC00346=-798156,-1296783
EC00347=-798156,-1296783
EC00348=-798156,-1296783
EC00349=-798156,-1296783
EC00350=-798156,-1296783
EC00351=-798156,-1296783
EC00352=-798156,-1296783
EC00353=-798156,-1296783
EC00354=-798156,-1296783
EC00355=-798156,-1296783
EC00356=-798156,-1296783
EC00357=-798156,-1296783
EC00358=-798156,-1296783
EC00359=-798156,-1296783
EC00360=-798156,-1296783
EC00361=-798156,-1296783
EC00362=-798156,-1296783
EC00363=-798156,-1296783
EC00364=-798156,-1296783
EC00365=-798156,-1296783
EC00366=-798156,-1296783
EC00367=-798156,-1296783
EC00368=-798156,-1296783
EC00369=-798156,-1296783
EC00370=-798156,-1296783
EC00371=-798156,-1296783
EC00372=-798156,-1296783
EC00373=-798156,-1296783
EC00374=-798156,-1296783
EC00375=-798156,-1296783
EC00376=-798156,-1296783
EC00377=-798156,-1296783
EC00378=-798156,-1296783
EC00379=-798156,-1296783
///POSTYPE BASE
///RECTAN
///RCONF 0,0,0,0,1,0,0,0,0,0,0,0,0,0,0,0,0,0,0,0,0,0,0,0
P00006=2.006,1.622,-0.565,0.0000,0.0000,0.0000
P00021=0.073,2.058,-0.109,0.0000,0.0000,0.0000
P00022=2.006,1.622,-0.565,0.0000,0.0000,0.0000
///RCONF 0,0,0,0,0,0,0,0,0,0,0,0,0,0,0,0,0,0,0,0,0,0,0,0
P00023=-2.957,-4.083,2.762,0.0000,0.0000,0.0000
P00024=-1.466,-0.226,-0.419,0.0000,0.0000,0.0000
P00025=3.643,0.007,-2.585,0.0000,0.0000,0.0000
P00026=2.644,0.055,-2.583,0.0000,0.0000,0.0000
P00027=2.278,0.099,-4.210,0.0000,0.0000,0.0000
P00028=-1.778,-0.182,-2.050,0.0000,0.0000,0.0000
P00029=1.749,4.006,-0.261,0.0000,0.0000,0.0000
P00032=-0.423,0.157,3.222,0.0000,0.0000,0.0000
P00033=0.854,-1.099,3.047,0.0000,0.0000,0.0000
///RCONF 0,0,0,0,1,0,0,0,0,0,0,0,0,0,0,0,0,0,0,0,0,0,0,0
P00034=-8.151,9.743,-4.393,0.0000,0.0000,0.0000
///RCONF 0,0,0,0,0,0,0,0,0,0,0,0,0,0,0,0,0,0,0,0,0,0,0,0
P00050=-0.123,2.174,-1.314,0.0000,0.0000,0.0000
P00051=-5.945,4.696,-10.293,0.0000,0.0000,0.0000
P00063=1197.217,207.358,-268.729,0.4863,35.2395,175.4586
P00099=-10.497,4.418,3.734,0.0000,0.0000,0.0000
//INST
///DATE 2024/12/09 16:48
///ATTR SC,RW
///GROUP1 RB1,BS1
///GROUP2 ST1
NOP
'X2_50&56B(90_180)
'Down
MOVJ C00000 BC00000 VJ=100.00  +MOVJ EC00000 VJ=100.00
MOVJ C00001 BC00001 VJ=100.00  +MOVJ EC00001 VJ=100.00
MOVJ C00002 BC00002 VJ=100.00  +MOVJ EC00002 VJ=100.00
'Path S4514
SFTOF3D
MOVJ C00003 BC00003 VJ=100.00  +MOVJ EC00003 VJ=100.00
MOVL C00004 BC00004 V=800.0  +MOVJ EC00004 VJ=100.00
SMOVL C00005 BC00005 V=166.7  +MOVJ EC00005
SREFP 3 C00006 BC00006  +REFP EC00006
CALL JOB:SEARCH-R1-S13D
SET P034 P006
SFTON3D P034
SMOVL C00007 BC00007 V=166.7  +MOVJ EC00007
SMOVL C00008 BC00008 V=166.7  +MOVJ EC00008
SMOVL C00009 BC00009 V=166.7  +MOVJ EC00009
SREFP 3 C00010 BC00010  +REFP EC00010
CALL JOB:SEARCH-R1-S13D
SET P034 P006
SFTON3D P034
SMOVL C00011 BC00011 V=166.7  +MOVJ EC00011
SMOVL C00012 BC00012 V=166.7  +MOVJ EC00012
SREFP 3 C00013 BC00013  +REFP EC00013
CALL JOB:SEARCH-R1-S13D
SET P034 P006
SFTON3D P034
SMOVL C00014 BC00014 V=166.7  +MOVJ EC00014
MOVL C00015 BC00015 V=1000.0  +MOVJ EC00015 VJ=100.00
'EndPath S4514
MOVJ C00016 BC00016 VJ=100.00  +MOVJ EC00016 VJ=100.00
MOVJ C00017 BC00017 VJ=100.00  +MOVJ EC00017 VJ=100.00
MOVJ C00018 BC00018 VJ=100.00  +MOVJ EC00018 VJ=100.00
MOVJ C00019 BC00019 VJ=100.00  +MOVJ EC00019 VJ=100.00
'Path S4515
SFTOF3D
MOVJ C00020 BC00020 VJ=100.00  +MOVJ EC00020 VJ=100.00
MOVL C00021 BC00021 V=800.0  +MOVJ EC00021 VJ=100.00
SMOVL C00022 BC00022 V=166.7  +MOVJ EC00022
SREFP 3 C00023 BC00023  +REFP EC00023
CALL JOB:SEARCH-R1-S13D
SET P033 P006
SFTON3D P033
SMOVL C00024 BC00024 V=250.0  +MOVJ EC00024
SMOVL C00025 BC00025 V=166.7  +MOVJ EC00025
SREFP 3 C00026 BC00026  +REFP EC00026
CALL JOB:SEARCH-R1-S13D
SET P033 P006
SFTON3D P033
SMOVL C00027 BC00027 V=166.7  +MOVJ EC00027
SMOVL C00028 BC00028 V=166.7  +MOVJ EC00028
SREFP 3 C00029 BC00029  +REFP EC00029
CALL JOB:SEARCH-R1-S13D
SET P033 P006
SFTON3D P033
SMOVL C00030 BC00030 V=166.7  +MOVJ EC00030
MOVL C00031 BC00031 V=1000.0  +MOVJ EC00031 VJ=100.00
'EndPath S4515
'Path S4516
SFTOF3D
MOVJ C00032 BC00032 VJ=100.00  +MOVJ EC00032 VJ=100.00
MOVL C00033 BC00033 V=800.0  +MOVJ EC00033 VJ=100.00
SMOVL C00034 BC00034 V=166.7  +MOVJ EC00034
SREFP 3 C00035 BC00035  +REFP EC00035
CALL JOB:SEARCH-R1-S13D
SET P032 P006
SFTON3D P032
SMOVL C00036 BC00036 V=166.7  +MOVJ EC00036
SMOVL C00037 BC00037 V=166.7  +MOVJ EC00037
SREFP 3 C00038 BC00038  +REFP EC00038
CALL JOB:SEARCH-R1-S13D
SET P032 P006
SFTON3D P032
SMOVL C00039 BC00039 V=166.7  +MOVJ EC00039
SMOVL C00040 BC00040 V=166.7  +MOVJ EC00040
SREFP 3 C00041 BC00041  +REFP EC00041
CALL JOB:SEARCH-R1-S13D
SET P032 P006
SFTON3D P032
SMOVL C00042 BC00042 V=166.7  +MOVJ EC00042
MOVL C00043 BC00043 V=1000.0  +MOVJ EC00043 VJ=100.00
'EndPath S4516
MOVJ C00044 BC00044 VJ=100.00  +MOVJ EC00044 VJ=100.00
MOVJ C00045 BC00045 VJ=100.00  +MOVJ EC00045 VJ=100.00
MOVL C00046 BC00046 V=800.0  +MOVJ EC00046 VJ=100.00
SMOVL C00047 BC00047 V=250.0  +MOVJ EC00047
SREFP 3 C00048 BC00048  +REFP EC00048
CALL JOB:SEARCH-R1-S13D
SET P099 P006
SFTON3D P099
SMOVL C00049 BC00049 V=166.7  +MOVJ EC00049
SMOVL C00050 BC00050 V=250.0  +MOVJ EC00050
SMOVL C00051 BC00051 V=166.7  +MOVJ EC00051
SREFP 3 C00052 BC00052  +REFP EC00052
CALL JOB:SEARCH-R1-S13D
SET P099 P006
SFTON3D P099
SMOVL C00053 BC00053 V=166.7  +MOVJ EC00053
SMOVL C00054 BC00054 V=800.0  +MOVJ EC00054
SFTOF3D
MOVJ C00055 BC00055 VJ=100.00  +MOVJ EC00055 VJ=100.00
'Path S4517
SFTOF3D
MOVJ C00056 BC00056 VJ=100.00  +MOVJ EC00056 VJ=100.00
'Path S4519
SFTOF3D
MOVJ C00057 BC00057 VJ=100.00  +MOVJ EC00057 VJ=100.00
MOVL C00058 BC00058 V=800.0  +MOVJ EC00058 VJ=100.00
SMOVL C00059 BC00059 V=166.7  +MOVJ EC00059
SREFP 3 C00060 BC00060  +REFP EC00060
CALL JOB:SEARCH-R1-S13D
SET P029 P006
SFTON3D P029
SMOVL C00061 BC00061 V=166.7  +MOVJ EC00061
SREFP 3 C00062 BC00062  +REFP EC00062
CALL JOB:SEARCH-R1-S13D
SET P029 P006
SFTON3D P029
SMOVL C00063 BC00063 V=166.7  +MOVJ EC00063
SFTOF3D
MOVL C00064 BC00064 V=800.0  +MOVJ EC00064 VJ=100.00
MOVL C00065 BC00065 V=1000.0  +MOVJ EC00065 VJ=100.00
SMOVL C00066 BC00066 V=250.0  +MOVJ EC00066
SMOVL C00067 BC00067 V=250.0  +MOVJ EC00067
SREFP 3 C00068 BC00068  +REFP EC00068
CALL JOB:SEARCH-R1-S13D
SET P050 P006
SFTON3D P050
SMOVL C00069 BC00069 V=166.7  +MOVJ EC00069
SREFP 3 C00070 BC00070  +REFP EC00070
CALL JOB:SEARCH-R1-S13D
SET P050 P006
SFTON3D P050
SMOVL C00071 BC00071 V=166.7  +MOVJ EC00071
SMOVL C00072 BC00072 V=250.0  +MOVJ EC00072
SMOVL C00073 BC00073 V=250.0  +MOVJ EC00073
SREFP 3 C00074 BC00074  +REFP EC00074
CALL JOB:SEARCH-R1-S13D
SET P050 P006
SFTON3D P050
SMOVL C00075 BC00075 V=166.7  +MOVJ EC00075
SFTOF3D
SMOVL C00076 BC00076 V=666.7  +MOVJ EC00076
SMOVL C00077 BC00077 V=666.7  +MOVJ EC00077
SMOVL C00078 BC00078 V=250.0  +MOVJ EC00078
SMOVL C00079 BC00079 V=250.0  +MOVJ EC00079
SREFP 3 C00080 BC00080  +REFP EC00080
CALL JOB:SEARCH-R1-S13D
SET P051 P006
SFTON3D P051
SMOVL C00081 BC00081 V=166.7  +MOVJ EC00081
SREFP 3 C00082 BC00082  +REFP EC00082
CALL JOB:SEARCH-R1-S13D
SET P051 P006
SFTON3D P051
SMOVL C00083 BC00083 V=250.0  +MOVJ EC00083
SMOVL C00084 BC00084 V=500.0  +MOVJ EC00084
SMOVL C00085 BC00085 V=250.0  +MOVJ EC00085
SREFP 3 C00086 BC00086  +REFP EC00086
CALL JOB:SEARCH-R1-S13D
SET P051 P006
SFTON3D P051
SMOVL C00087 BC00087 V=166.7  +MOVJ EC00087
SFTOF3D
SMOVL C00088 BC00088 V=666.7  +MOVJ EC00088
'EndPath S4519
MOVJ C00089 BC00089 VJ=100.00  +MOVJ EC00089 VJ=100.00
'Path S4520
SFTOF3D
MOVJ C00090 BC00090 VJ=100.00  +MOVJ EC00090 VJ=100.00
MOVL C00091 BC00091 V=800.0  +MOVJ EC00091 VJ=100.00
SMOVL C00092 BC00092 V=133.3  +MOVJ EC00092
SREFP 3 C00093 BC00093  +REFP EC00093
CALL JOB:SEARCH-R1-S13D
SET P028 P006
SFTON3D P028
SMOVL C00094 BC00094 V=166.7  +MOVJ EC00094
SMOVL C00095 BC00095 V=166.7  +MOVJ EC00095
SREFP 3 C00096 BC00096  +REFP EC00096
CALL JOB:SEARCH-R1-S13D
SET P028 P006
SFTON3D P028
SMOVL C00097 BC00097 V=166.7  +MOVJ EC00097
MOVL C00098 BC00098 V=800.0  +MOVJ EC00098 VJ=100.00
MOVL C00099 BC00099 V=1000.0  +MOVJ EC00099 VJ=100.00
'EndPath S4520
'Path S4521
SFTOF3D
MOVJ C00100 BC00100 VJ=100.00  +MOVJ EC00100 VJ=100.00
MOVL C00101 BC00101 V=800.0  +MOVJ EC00101 VJ=100.00
SMOVL C00102 BC00102 V=166.7  +MOVJ EC00102
SREFP 3 C00103 BC00103  +REFP EC00103
CALL JOB:SEARCH-R1-S13D
SET P027 P006
SFTON3D P027
SMOVL C00104 BC00104 V=166.7  +MOVJ EC00104
SMOVL C00105 BC00105 V=166.7  +MOVJ EC00105
SREFP 3 C00106 BC00106  +REFP EC00106
CALL JOB:SEARCH-R1-S13D
SET P027 P006
SFTON3D P027
SMOVL C00107 BC00107 V=166.7  +MOVJ EC00107
MOVL C00108 BC00108 V=800.0  +MOVJ EC00108 VJ=100.00
MOVL C00109 BC00109 V=1000.0  +MOVJ EC00109 VJ=100.00
'EndPath S4521
MOVJ C00110 BC00110 VJ=100.00  +MOVJ EC00110 VJ=100.00
'Up
MOVJ C00111 BC00111 VJ=100.00  +MOVJ EC00111 VJ=100.00
MOVJ C00112 BC00112 VJ=100.00  +MOVJ EC00112 VJ=100.00
'Path S4522
SFTOF3D
MOVJ C00113 BC00113 VJ=100.00  +MOVJ EC00113 VJ=100.00
MOVL C00114 BC00114 V=800.0  +MOVJ EC00114 VJ=100.00
SMOVL C00115 BC00115 V=166.7  +MOVJ EC00115
SREFP 3 C00116 BC00116  +REFP EC00116
CALL JOB:SEARCH-R1-S13D
SET P026 P006
SFTON3D P026
SMOVL C00117 BC00117 V=166.7  +MOVJ EC00117
SREFP 3 C00118 BC00118  +REFP EC00118
CALL JOB:SEARCH-R1-S13D
SET P026 P006
SFTON3D P026
SMOVL C00119 BC00119 V=166.7  +MOVJ EC00119
MOVL C00120 BC00120 V=1000.0  +MOVJ EC00120 VJ=100.00
'EndPath S4522
'Path S4523
SFTOF3D
MOVJ C00121 BC00121 VJ=100.00  +MOVJ EC00121 VJ=100.00
MOVL C00122 BC00122 V=800.0  +MOVJ EC00122 VJ=100.00
SMOVL C00123 BC00123 V=166.7  +MOVJ EC00123
SREFP 3 C00124 BC00124  +REFP EC00124
CALL JOB:SEARCH-R1-S13D
SET P025 P006
SFTON3D P025
SMOVL C00125 BC00125 V=166.7  +MOVJ EC00125
SREFP 3 C00126 BC00126  +REFP EC00126
CALL JOB:SEARCH-R1-S13D
SET P025 P006
SFTON3D P025
SMOVL C00127 BC00127 V=166.7  +MOVJ EC00127
SMOVL C00128 BC00128 V=166.7  +MOVJ EC00128
SMOVL C00129 BC00129 V=166.7  +MOVJ EC00129
SREFP 3 C00130 BC00130  +REFP EC00130
CALL JOB:SEARCH-R1-S13D
SET P025 P006
SFTON3D P025
SMOVL C00131 BC00131 V=166.7  +MOVJ EC00131
MOVL C00132 BC00132 V=1000.0  +MOVJ EC00132 VJ=100.00
'EndPath S4523
'Path S4524
SFTOF3D
MOVJ C00133 BC00133 VJ=100.00  +MOVJ EC00133 VJ=100.00
MOVL C00134 BC00134 V=800.0  +MOVJ EC00134 VJ=100.00
SMOVL C00135 BC00135 V=166.7  +MOVJ EC00135
SREFP 3 C00136 BC00136  +REFP EC00136
CALL JOB:SEARCH-R1-S13D
SET P024 P006
SFTON3D P024
SMOVL C00137 BC00137 V=166.7  +MOVJ EC00137
SREFP 3 C00138 BC00138  +REFP EC00138
CALL JOB:SEARCH-R1-S13D
SET P024 P006
SFTON3D P024
SMOVL C00139 BC00139 V=166.7  +MOVJ EC00139
SMOVL C00140 BC00140 V=166.7  +MOVJ EC00140
SREFP 3 C00141 BC00141  +REFP EC00141
CALL JOB:SEARCH-R1-S13D
SET P024 P006
SFTON3D P024
SMOVL C00142 BC00142 V=166.7  +MOVJ EC00142
MOVL C00143 BC00143 V=1000.0  +MOVJ EC00143 VJ=100.00
'EndPath S4524
'Path S4525
SFTOF3D
MOVJ C00144 BC00144 VJ=100.00  +MOVJ EC00144 VJ=100.00
MOVL C00145 BC00145 V=800.0  +MOVJ EC00145 VJ=100.00
SMOVL C00146 BC00146 V=166.7  +MOVJ EC00146
SREFP 3 C00147 BC00147  +REFP EC00147
CALL JOB:SEARCH-R1-S13D
SET P023 P006
SFTON3D P023
SMOVL C00148 BC00148 V=166.7  +MOVJ EC00148
SREFP 3 C00149 BC00149  +REFP EC00149
CALL JOB:SEARCH-R1-S13D
SET P023 P006
SFTON3D P023
SMOVL C00150 BC00150 V=166.7  +MOVJ EC00150
SMOVL C00151 BC00151 V=166.7  +MOVJ EC00151
SREFP 3 C00152 BC00152  +REFP EC00152
CALL JOB:SEARCH-R1-S13D
SET P023 P006
SFTON3D P023
SMOVL C00153 BC00153 V=166.7  +MOVJ EC00153
MOVL C00154 BC00154 V=1000.0  +MOVJ EC00154 VJ=100.00
'EndPath S4525
'Path S4729
SFTOF3D
MOVJ C00155 BC00155 VJ=100.00  +MOVJ EC00155 VJ=100.00
MOVL C00156 BC00156 V=800.0  +MOVJ EC00156 VJ=100.00
SMOVL C00157 BC00157 V=166.7  +MOVJ EC00157
SREFP 3 C00158 BC00158  +REFP EC00158
CALL JOB:SEARCH-R1-S13D
SET P063 P006
SFTON3D P063
SMOVL C00159 BC00159 V=166.7  +MOVJ EC00159
SREFP 3 C00160 BC00160  +REFP EC00160
CALL JOB:SEARCH-R1-S13D
SET P063 P006
SFTON3D P063
SMOVL C00161 BC00161 V=166.7  +MOVJ EC00161
SMOVL C00162 BC00162 V=166.7  +MOVJ EC00162
SREFP 3 C00163 BC00163  +REFP EC00163
CALL JOB:SEARCH-R1-S13D
SET P063 P006
SFTON3D P063
SMOVL C00164 BC00164 V=166.7  +MOVJ EC00164
MOVL C00165 BC00165 V=1000.0  +MOVJ EC00165 VJ=100.00
'EndPath S4729
'Path S4526
SFTOF3D
MOVJ C00166 BC00166 VJ=100.00  +MOVJ EC00166 VJ=100.00
MOVL C00167 BC00167 V=800.0  +MOVJ EC00167 VJ=100.00
SMOVL C00168 BC00168 V=166.7  +MOVJ EC00168
SREFP 3 C00169 BC00169  +REFP EC00169
CALL JOB:SEARCH-R1-S13D
SET P022 P006
SFTON3D P022
SMOVL C00170 BC00170 V=166.7  +MOVJ EC00170
SREFP 3 C00171 BC00171  +REFP EC00171
CALL JOB:SEARCH-R1-S13D
SET P022 P006
SFTON3D P022
SMOVL C00172 BC00172 V=166.7  +MOVJ EC00172
SREFP 3 C00173 BC00173  +REFP EC00173
CALL JOB:SEARCH-R1-S13D
SET P022 P006
SFTON3D P022
SMOVL C00174 BC00174 V=166.7  +MOVJ EC00174
MOVL C00175 BC00175 V=1000.0  +MOVJ EC00175 VJ=100.00
'EndPath S4526
'Path S4527
SFTOF3D
MOVJ C00176 BC00176 VJ=100.00  +MOVJ EC00176 VJ=100.00
MOVL C00177 BC00177 V=800.0  +MOVJ EC00177 VJ=100.00
SMOVL C00178 BC00178 V=166.7  +MOVJ EC00178
SREFP 3 C00179 BC00179  +REFP EC00179
CALL JOB:SEARCH-R1-S13D
SET P021 P006
SFTON3D P021
SMOVL C00180 BC00180 V=166.7  +MOVJ EC00180
SREFP 3 C00181 BC00181  +REFP EC00181
CALL JOB:SEARCH-R1-S13D
SET P021 P006
SFTON3D P021
SMOVL C00182 BC00182 V=250.0  +MOVJ EC00182
SMOVL C00183 BC00183 V=166.7  +MOVJ EC00183
SREFP 3 C00184 BC00184  +REFP EC00184
CALL JOB:SEARCH-R1-S13D
SET P021 P006
SFTON3D P021
SMOVL C00185 BC00185 V=166.7  +MOVJ EC00185
MOVL C00186 BC00186 V=1000.0  +MOVJ EC00186 VJ=100.00
'EndPath S4527
MOVJ C00187 BC00187 VJ=100.00  +MOVJ EC00187 VJ=100.00
'Path W4730
SFTOF3D
SFTON3D P024
MOVJ C00188 BC00188 VJ=100.00  +MOVJ EC00188 VJ=100.00
SMOVL C00189 BC00189 V=800.0  +MOVJ EC00189
SMOVL C00190 BC00190 V=150.0 PL=0  +MOVJ EC00190
MACRO1 MJ#(0) ARGF14
ARCON
SMOVL C00191 BC00191 V=10.0  +MOVJ EC00191
SMOVL C00192 BC00192 V=11.7  +MOVJ EC00192
ARCOF
SMOVL C00193 BC00193 V=800.0  +MOVJ EC00193
SMOVL C00194 BC00194 V=1000.0  +MOVJ EC00194
SFTOF3D
'EndPath W4730
MOVJ C00195 BC00195 VJ=100.00  +MOVJ EC00195 VJ=100.00
'Path W4731
SFTOF3D
SFTON3D P063
MOVJ C00196 BC00196 VJ=100.00  +MOVJ EC00196 VJ=100.00
SMOVL C00197 BC00197 V=800.0  +MOVJ EC00197
SMOVL C00198 BC00198 V=150.0 PL=0  +MOVJ EC00198
MACRO1 MJ#(0) ARGF9
ARCON
SMOVL C00199 BC00199 V=10.0  +MOVJ EC00199
SMOVL C00200 BC00200 V=10.0  +MOVJ EC00200
ARCOF
SMOVL C00201 BC00201 V=800.0  +MOVJ EC00201
SMOVL C00202 BC00202 V=1000.0  +MOVJ EC00202
SFTOF3D
'EndPath W4731
'Path W4528
SFTOF3D
SFTON3D P021
MOVJ C00203 BC00203 VJ=100.00  +MOVJ EC00203 VJ=100.00
SMOVL C00204 BC00204 V=800.0  +MOVJ EC00204
SMOVL C00205 BC00205 V=166.7 PL=0  +MOVJ EC00205
MACRO1 MJ#(0) ARGF21
ARCON
SMOVL C00206 BC00206 V=10.8  +MOVJ EC00206
SFTON3D P022
SMOVL C00207 BC00207 V=10.8  +MOVJ EC00207
SMOVL C00208 BC00208 V=10.8  +MOVJ EC00208
ARCOF
SMOVL C00209 BC00209 V=800.0  +MOVJ EC00209
SMOVL C00210 BC00210 V=1000.0  +MOVJ EC00210
SFTOF3D
'EndPath W4528
'Path W4529
SFTOF3D
SFTON3D P022
MOVJ C00211 BC00211 VJ=100.00  +MOVJ EC00211 VJ=100.00
SMOVL C00212 BC00212 V=800.0  +MOVJ EC00212
SMOVL C00213 BC00213 V=166.7 PL=0  +MOVJ EC00213
ARCON
SMOVL C00214 BC00214 V=10.8  +MOVJ EC00214
ARCOF
SMOVL C00215 BC00215 V=800.0  +MOVJ EC00215
SMOVL C00216 BC00216 V=1000.0  +MOVJ EC00216
SFTOF3D
'EndPath W4529
'Path W4530
SFTOF3D
SFTON3D P023
MOVJ C00217 BC00217 VJ=100.00  +MOVJ EC00217 VJ=100.00
SMOVL C00218 BC00218 V=800.0  +MOVJ EC00218
SMOVL C00219 BC00219 V=166.7 PL=0  +MOVJ EC00219
ARCON
SWVON WEV#(60)
SMOVL C00220 BC00220 V=7.5  +MOVJ EC00220
SFTON3D P024
SMOVL C00221 BC00221 V=7.5  +MOVJ EC00221
SMOVL C00222 BC00222 V=7.5  +MOVJ EC00222
ARCOF
SWVOF
SMOVL C00223 BC00223 V=800.0  +MOVJ EC00223
SMOVL C00224 BC00224 V=1000.0  +MOVJ EC00224
SFTOF3D
'EndPath W4530
'Path W4531
SFTOF3D
SFTON3D P025
MOVJ C00225 BC00225 VJ=100.00  +MOVJ EC00225 VJ=100.00
SMOVL C00226 BC00226 V=800.0  +MOVJ EC00226
SMOVL C00227 BC00227 V=166.7 PL=0  +MOVJ EC00227
ARCON
SMOVL C00228 BC00228 V=10.8  +MOVJ EC00228
SFTON3D P026
SMOVL C00229 BC00229 V=10.8  +MOVJ EC00229
SMOVL C00230 BC00230 V=10.8  +MOVJ EC00230
ARCOF
SMOVL C00231 BC00231 V=800.0  +MOVJ EC00231
SMOVL C00232 BC00232 V=1000.0  +MOVJ EC00232
SFTOF3D
'EndPath W4531
'Down
MOVJ C00233 BC00233 VJ=100.00  +MOVJ EC00233 VJ=100.00
MOVJ C00234 BC00234 VJ=100.00  +MOVJ EC00234 VJ=100.00
MOVJ C00235 BC00235 VJ=100.00  +MOVJ EC00235 VJ=100.00
MOVJ C00236 BC00236 VJ=100.00  +MOVJ EC00236 VJ=100.00
'Path W4532
SFTOF3D
MOVJ C00237 BC00237 VJ=100.00  +MOVJ EC00237 VJ=100.00
MOVJ C00238 BC00238 VJ=100.00  +MOVJ EC00238 VJ=100.00
'Path W4534
SFTOF3D
SFTON3D P033
MOVJ C00239 BC00239 VJ=100.00  +MOVJ EC00239 VJ=100.00
SMOVL C00240 BC00240 V=800.0  +MOVJ EC00240
SMOVL C00241 BC00241 V=166.7 PL=0  +MOVJ EC00241
MACRO1 MJ#(0) ARGF14
ARCON
SMOVL C00242 BC00242 V=10.0  +MOVJ EC00242
SMOVL C00243 BC00243 V=10.0  +MOVJ EC00243
SMOVL C00244 BC00244 V=10.0  +MOVJ EC00244
ARCOF
SMOVL C00245 BC00245 V=800.0  +MOVJ EC00245
SMOVL C00246 BC00246 V=166.7  +MOVJ EC00246
SMOVL C00247 BC00247 V=166.7  +MOVJ EC00247
ARCON
SMOVL C00248 BC00248 V=13.3  +MOVJ EC00248
SMOVL C00249 BC00249 V=13.3  +MOVJ EC00249
ARCOF
SMOVL C00250 BC00250 V=166.7  +MOVJ EC00250
SMOVL C00251 BC00251 V=500.0  +MOVJ EC00251
SMOVL C00252 BC00252 V=133.3  +MOVJ EC00252
ARCON
SMOVL C00253 BC00253 V=13.3  +MOVJ EC00253
SMOVL C00254 BC00254 V=13.3  +MOVJ EC00254
ARCOF
SMOVL C00255 BC00255 V=250.0  +MOVJ EC00255
SMOVL C00256 BC00256 V=1000.0  +MOVJ EC00256
SFTOF3D
'EndPath W4534
'Path W4535
SFTOF3D
SFTON3D P032
MOVJ C00257 BC00257 VJ=100.00  +MOVJ EC00257 VJ=100.00
SMOVL C00258 BC00258 V=800.0  +MOVJ EC00258
SMOVL C00259 BC00259 V=166.7 PL=0  +MOVJ EC00259
ARCON
SMOVL C00260 BC00260 V=10.0  +MOVJ EC00260
SMOVL C00261 BC00261 V=10.0  +MOVJ EC00261
SMOVL C00262 BC00262 V=11.7  +MOVJ EC00262
ARCOF
SMOVL C00263 BC00263 V=800.0  +MOVJ EC00263
SMOVL C00264 BC00264 V=250.0  +MOVJ EC00264
SMOVL C00265 BC00265 V=166.7  +MOVJ EC00265
ARCON
SMOVL C00266 BC00266 V=10.8  +MOVJ EC00266
ARCOF
SMOVL C00267 BC00267 V=250.0  +MOVJ EC00267
SMOVL C00268 BC00268 V=1000.0  +MOVJ EC00268
SFTOF3D
'EndPath W4535
'Path W4536
SFTOF3D
SFTON3D P032
MOVJ C00269 BC00269 VJ=100.00  +MOVJ EC00269 VJ=100.00
SFTOF3D
'EndPath W4536
MOVJ C00270 BC00270 VJ=100.00  +MOVJ EC00270 VJ=100.00
'Path W4537
SFTOF3D
SFTON3D P027
MOVJ C00271 BC00271 VJ=100.00  +MOVJ EC00271 VJ=100.00
SMOVL C00272 BC00272 V=800.0  +MOVJ EC00272
SMOVL C00273 BC00273 V=150.0 PL=0  +MOVJ EC00273
MACRO1 MJ#(0) ARGF9
ARCON
SMOVL C00274 BC00274 V=10.8  +MOVJ EC00274
SMOVL C00275 BC00275 V=10.8  +MOVJ EC00275
ARCOF
SMOVL C00276 BC00276 V=800.0  +MOVJ EC00276
SMOVL C00277 BC00277 V=1000.0  +MOVJ EC00277
SFTOF3D
'EndPath W4537
'Path W4538
SFTOF3D
SFTON3D P027
SMOVL C00278 BC00278 V=1000.0  +MOVJ EC00278
SMOVL C00279 BC00279 V=150.0 PL=0  +MOVJ EC00279
ARCON
SMOVL C00280 BC00280 V=10.8  +MOVJ EC00280
ARCOF
SMOVL C00281 BC00281 V=800.0  +MOVJ EC00281
SFTOF3D
'EndPath W4538
'Path W4539
SFTOF3D
SFTON3D P028
SMOVL C00282 BC00282 V=1000.0  +MOVJ EC00282
SMOVL C00283 BC00283 V=150.0 PL=0  +MOVJ EC00283
ARCON
SMOVL C00284 BC00284 V=10.8  +MOVJ EC00284
ARCOF
SMOVL C00285 BC00285 V=800.0  +MOVJ EC00285
SFTOF3D
'EndPath W4539
'Path W4540
SFTOF3D
SFTON3D P028
SMOVL C00286 BC00286 V=1000.0  +MOVJ EC00286
SMOVL C00287 BC00287 V=150.0 PL=0  +MOVJ EC00287
ARCON
SMOVL C00288 BC00288 V=10.8  +MOVJ EC00288
SMOVL C00289 BC00289 V=10.8  +MOVJ EC00289
ARCOF
SMOVL C00290 BC00290 V=800.0  +MOVJ EC00290
SMOVL C00291 BC00291 V=1000.0  +MOVJ EC00291
SFTOF3D
'EndPath W4540
MOVJ C00292 BC00292 VJ=100.00  +MOVJ EC00292 VJ=100.00
MOVJ C00293 BC00293 VJ=100.00  +MOVJ EC00293 VJ=100.00
SMOVL C00294 BC00294 V=666.7  +MOVJ EC00294
MACRO1 MJ#(0) ARGF14
SFTON3D P051
SMOVL C00295 BC00295 V=166.7  +MOVJ EC00295
ARCON
SMOVL C00296 BC00296 V=10.8  +MOVJ EC00296
ARCOF
SMOVL C00297 BC00297 V=133.3  +MOVJ EC00297
SMOVL C00298 BC00298 V=133.3  +MOVJ EC00298
ARCON
SMOVL C00299 BC00299 V=6.7  +MOVJ EC00299
ARCOF
SMOVL C00300 BC00300 V=133.3  +MOVJ EC00300
SMOVL C00301 BC00301 V=250.0  +MOVJ EC00301
MACRO1 MJ#(0) ARGF9
SMOVL C00302 BC00302 V=133.3  +MOVJ EC00302
ARCON
SMOVL C00303 BC00303 V=8.3  +MOVJ EC00303
ARCOF
SMOVL C00304 BC00304 V=250.0  +MOVJ EC00304
SMOVL C00305 BC00305 V=250.0  +MOVJ EC00305
MACRO1 MJ#(0) ARGF14
SMOVL C00306 BC00306 V=166.7  +MOVJ EC00306
ARCON
SMOVL C00307 BC00307 V=10.8  +MOVJ EC00307
ARCOF
SMOVL C00308 BC00308 V=166.7  +MOVJ EC00308
SFTON3D P050
SMOVL C00309 BC00309 V=166.7  +MOVJ EC00309
ARCON
SMOVL C00310 BC00310 V=10.8  +MOVJ EC00310
ARCOF
SMOVL C00311 BC00311 V=166.7  +MOVJ EC00311
ARCON
SMOVL C00312 BC00312 V=11.7  +MOVJ EC00312
SMOVL C00313 BC00313 V=11.7  +MOVJ EC00313
ARCOF
SMOVL C00314 BC00314 V=33.3  +MOVJ EC00314
SMOVL C00315 BC00315 V=33.3  +MOVJ EC00315
ARCON
SMOVL C00316 BC00316 V=11.7  +MOVJ EC00316
ARCOF
SMOVL C00317 BC00317 V=166.7  +MOVJ EC00317
SFTOF3D
MOVJ C00318 BC00318 VJ=100.00  +MOVJ EC00318 VJ=100.00
'Path W4541
SFTOF3D
SFTON3D P029
MOVJ C00319 BC00319 VJ=100.00  +MOVJ EC00319 VJ=100.00
SMOVL C00320 BC00320 V=800.0  +MOVJ EC00320
MACRO1 MJ#(0) ARGF9
SMOVL C00321 BC00321 V=150.0 PL=0  +MOVJ EC00321
ARCON
SMOVL C00322 BC00322 V=10.8  +MOVJ EC00322
ARCOF
SMOVL C00323 BC00323 V=800.0  +MOVJ EC00323
SMOVL C00324 BC00324 V=1000.0  +MOVJ EC00324
SFTOF3D
'EndPath W4541
'Path W4542
SFTOF3D
SFTON3D P029
MOVJ C00325 BC00325 VJ=100.00  +MOVJ EC00325 VJ=100.00
SMOVL C00326 BC00326 V=800.0  +MOVJ EC00326
SMOVL C00327 BC00327 V=150.0 PL=0  +MOVJ EC00327
ARCON
SMOVL C00328 BC00328 V=10.8  +MOVJ EC00328
ARCOF
SMOVL C00329 BC00329 V=800.0  +MOVJ EC00329
SMOVL C00330 BC00330 V=1000.0  +MOVJ EC00330
SFTOF3D
'EndPath W4542
MOVJ C00331 BC00331 VJ=100.00  +MOVJ EC00331 VJ=100.00
MOVJ C00332 BC00332 VJ=100.00  +MOVJ EC00332 VJ=100.00
MOVJ C00333 BC00333 VJ=100.00  +MOVJ EC00333 VJ=100.00
MOVJ C00334 BC00334 VJ=100.00  +MOVJ EC00334 VJ=100.00
SFTON3D P099
SMOVL C00335 BC00335 V=166.7  +MOVJ EC00335
ARCON
SMOVL C00336 BC00336 V=10.8  +MOVJ EC00336
ARCOF
SFTOF3D
SMOVL C00337 BC00337 V=166.7  +MOVJ EC00337
MOVJ C00338 BC00338 VJ=100.00  +MOVJ EC00338 VJ=100.00
MOVJ C00339 BC00339 VJ=100.00  +MOVJ EC00339 VJ=100.00
MOVJ C00340 BC00340 VJ=100.00  +MOVJ EC00340 VJ=100.00
MOVJ C00341 BC00341 VJ=100.00  +MOVJ EC00341 VJ=100.00
SFTON3D P050
SMOVL C00342 BC00342 V=166.7  +MOVJ EC00342
ARCON
SMOVL C00343 BC00343 V=11.7  +MOVJ EC00343
ARCOF
SMOVL C00344 BC00344 V=133.3  +MOVJ EC00344
SMOVL C00345 BC00345 V=133.3  +MOVJ EC00345
SMOVL C00346 BC00346 V=133.3  +MOVJ EC00346
ARCON
SMOVL C00347 BC00347 V=10.8  +MOVJ EC00347
ARCOF
SMOVL C00348 BC00348 V=416.7  +MOVJ EC00348
SFTOF3D
MOVJ C00349 BC00349 VJ=100.00  +MOVJ EC00349 VJ=100.00
MOVJ C00350 BC00350 VJ=100.00  +MOVJ EC00350 VJ=100.00
MOVJ C00351 BC00351 VJ=100.00  +MOVJ EC00351 VJ=100.00
SFTON3D P032
SMOVL C00352 BC00352 V=133.3  +MOVJ EC00352
ARCON
SMOVL C00353 BC00353 V=13.3  +MOVJ EC00353
SMOVL C00354 BC00354 V=13.3  +MOVJ EC00354
SMOVL C00355 BC00355 V=13.3  +MOVJ EC00355
ARCOF
SMOVL C00356 BC00356 V=250.0  +MOVJ EC00356
SMOVL C00357 BC00357 V=666.7  +MOVJ EC00357
MOVJ C00358 BC00358 VJ=100.00  +MOVJ EC00358 VJ=100.00
MOVJ C00359 BC00359 VJ=100.00  +MOVJ EC00359 VJ=100.00
'Path W4543
SFTOF3D
SFTON3D P034
MOVJ C00360 BC00360 VJ=100.00  +MOVJ EC00360 VJ=100.00
SMOVL C00361 BC00361 V=800.0  +MOVJ EC00361
SMOVL C00362 BC00362 V=150.0 PL=0  +MOVJ EC00362
MACRO1 MJ#(0) ARGF14
ARCON
SMOVL C00363 BC00363 V=10.8  +MOVJ EC00363
SMOVL C00364 BC00364 V=10.8  +MOVJ EC00364
ARCOF
SMOVL C00365 BC00365 V=800.0  +MOVJ EC00365
SMOVL C00366 BC00366 V=333.3  +MOVJ EC00366
SMOVL C00367 BC00367 V=133.3  +MOVJ EC00367
ARCON
SMOVL C00368 BC00368 V=10.8  +MOVJ EC00368
SMOVL C00369 BC00369 V=10.8  +MOVJ EC00369
ARCOF
SMOVL C00370 BC00370 V=166.7  +MOVJ EC00370
SMOVL C00371 BC00371 V=166.7  +MOVJ EC00371
SMOVL C00372 BC00372 V=166.7  +MOVJ EC00372
SMOVL C00373 BC00373 V=166.7  +MOVJ EC00373
ARCON
SMOVL C00374 BC00374 V=10.8  +MOVJ EC00374
ARCOF
SMOVL C00375 BC00375 V=166.7  +MOVJ EC00375
SMOVL C00376 BC00376 V=166.7  +MOVJ EC00376
MOVJ C00377 BC00377 VJ=30.00  +MOVJ EC00377 VJ=100.00
SFTOF3D
'EndPath W4543
MOVJ C00378 BC00378 VJ=100.00  +MOVJ EC00378 VJ=100.00
MOVJ C00379 BC00379 VJ=100.00  +MOVJ EC00379 VJ=100.00
END
